PROGRAM AP_1
VAR
	GetPlate			:Seq_Get_plate;
	SetPlate1			:Seq_Set_Plate_1;
END_VAR

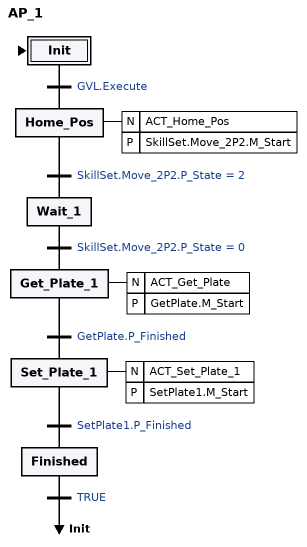
INITIAL_STEP Init:
END_STEP
TRANSITION FROM Init TO Home_Pos
    := GVL.Execute;
END_TRANSITION
STEP Home_Pos:
    ACT_Home_Pos(N);
    SkillSet.Move_2P2.M_Start(P);
END_STEP
TRANSITION FROM Home_Pos TO Wait_1
    := SkillSet.Move_2P2.P_State = 2;
END_TRANSITION
STEP Wait_1:
END_STEP
TRANSITION FROM Wait_1 TO Get_Plate_1
    := SkillSet.Move_2P2.P_State = 0;
END_TRANSITION
STEP Get_Plate_1:
    ACT_Get_Plate(N);
    GetPlate.M_Start(P);
END_STEP
TRANSITION FROM Get_Plate_1 TO Set_Plate_1
    := GetPlate.P_Finished;
END_TRANSITION
STEP Set_Plate_1:
    ACT_Set_Plate_1(N);
    SetPlate1.M_Start(P);
END_STEP
TRANSITION FROM Set_Plate_1 TO Finished
    := SetPlate1.P_Finished;
END_TRANSITION
STEP Finished:
END_STEP
TRANSITION FROM Finished TO Init
    := TRUE;
END_TRANSITION

ACTION ACT_Get_Plate:
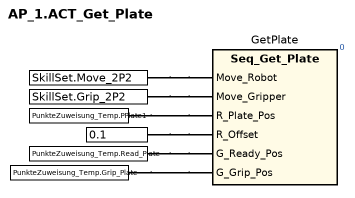
GetPlate(
    Move_Robot := SkillSet.Move_2P2,
    Move_Gripper := SkillSet.Grip_2P2,
    R_Plate_Pos := PunkteZuweisung_Temp.PPlate1,
    R_Offset := 0.1,
    G_Ready_Pos := PunkteZuweisung_Temp.Read_Plate,
    G_Grip_Pos := PunkteZuweisung_Temp.Grip_Plate); // Seq_Get_Plate
END_ACTION

ACTION ACT_Home_Pos:
SkillSet.Move_2P2.P_Prozessparameter := PunkteZuweisung_Temp.PHome;
END_ACTION

ACTION ACT_Set_Plate_1:
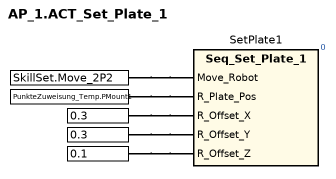
SetPlate1(
    Move_Robot := SkillSet.Move_2P2,
    R_Plate_Pos := PunkteZuweisung_Temp.PMount1,
    R_Offset_X := 0.3,
    R_Offset_Y := 0.3,
    R_Offset_Z := 0.1); // Seq_Set_Plate_1
END_ACTION

END_PROGRAM

(* stored: Version 1.1.0.1
   POU AP_1: Id {1ec52e47-a75e-409f-9983-fd458e25da35}, SpecialFunc None
   Folder 01_Zuweisung: Id {f23edcfb-a572-4ff4-bf31-505b6a2c49a1}
   Action ACT_Get_Plate: Id {5ae96c55-97e8-41b8-bb9e-45111a22ef81}
   Action ACT_Home_Pos: Id {59404226-b6e6-4ec2-9b80-1c584e73659b}
   Action ACT_Set_Plate_1: Id {87c2d091-e350-4806-a438-898c82624f6d} *)
